{attribute 'qualified_only'}
{attribute 'strict'}
TYPE E_CanItfHelperHResult :
(
	NoError 						:= 0,  // values >= 0 implies no error and/or informational. values < 0 implies error. 
	
	InvalidSetup 					:= -1, //pointers to ST_CanQueue are zero or sizeof ST_CanQueue doesn't equal 11bit or 29bit version.
	InvalidPointer					:= -2, //pointer parameter is zero.
	
	RxQueueHasUnreadMessages 		:= -100, // Rx Queue 'NoOfRxMessages' not equal RxMessagesAckedCnt, call either mGetRxMessages or mAckRxMessages.
	RxQueueEmpty 					:= -101, // Rx queue is empty, wait for more data.
	NoNewRxMessages 				:= -102, // Rx queue has not received new data yet.
	RxMessageInvalid				:= -103, // Rx Message returned is invalid, ignore result. Re-read Rx Messages.

	TxQueueFull 					:= -200, //NumOfMessages variable in Tx Queue is at or is greater then the allowed amount. Call aResetTxQueue and refill queue.
	TxQueueEmpty 					:= -201, // Tx queue 'NoOfTxMessages' value is zero, use mAddTxMessage to add messages.
	TxQueueInvalid					:= -202, //Tx Queue
	TxQueueIsBusy					:= -203 // Tx queue 'TxCounter' and Rx queue 'TxCounter' are not equal, waiting for CanInterface to send previous messages.
	
)DINT;
END_TYPE

(* stored: Version 1.1.0.1, ProductVersion 3.1.4024.11
   DUT E_CanItfHelperHResult: Id {1ef838dd-b8aa-4550-b34e-5c2faaaad70c} *)
